PROGRAM PRG_07_Servo
VAR
	fbMC_Power_Ax1: MC_Power;
	fbMC_Power_Ax2: MC_Power;
	fbMC_Jog_Ax1: MC_Jog;
	fbMC_Jog_Ax2: MC_Jog;
	fbMC_Reset_Ax1: MC_Reset;
	fbMC_Reset_Ax2: MC_Reset;
	fbMC_Stop_Ax1: MC_Stop;
	fbMC_Stop_Ax2: MC_Stop;
	
	rJogSpeed:	REAL;
	
	bTest1: BOOL;
	MC_ReadStatus_0: MC_ReadStatus;
	MC_ReadStatus_1: MC_ReadStatus;
	R_TRIG_0: R_TRIG;
	R_TRIG_1: R_TRIG;
	MC_MoveVelocity_0: MC_MoveVelocity;
	uAx1Encoder: UDINT;
	bJogSpeedChange: BOOL;
	t_JogSpeedChange: TP;
	JogSpeegTrig: F_TRIG;
	iPowerOverride: INT;
	tof_SawDownLimit: TOF;
	TRIG_SawDownLimit: r_trig;
	SR_SawDownLimit: SR;

	ton_SawDownLimitTimer: ton;
	SR_ZAxisBuffer: SR;
	F_TRIG_ZAxisCapturedValue: F_TRIG;
	rZAxisBufferSpeed: REAL;
	rZAxisSlowSpeed: REAL;
	rZAxisMedSpeed: REAL;
	rZAxisFastSpeed: REAL;
	sr_ZAxisBufferZone: SR;
	rZAxisCurrentFeedbackSpeed: REAL;
	F_TRIG_ZAxisUpperLimitValue: F_TRIG;
	F_TRIG_ZAxisLowerLimitValue: F_TRIG;
	iZAxisCapturedBufferValue: DINT;

END_VAR

ACTION ACT_07_1_Power:
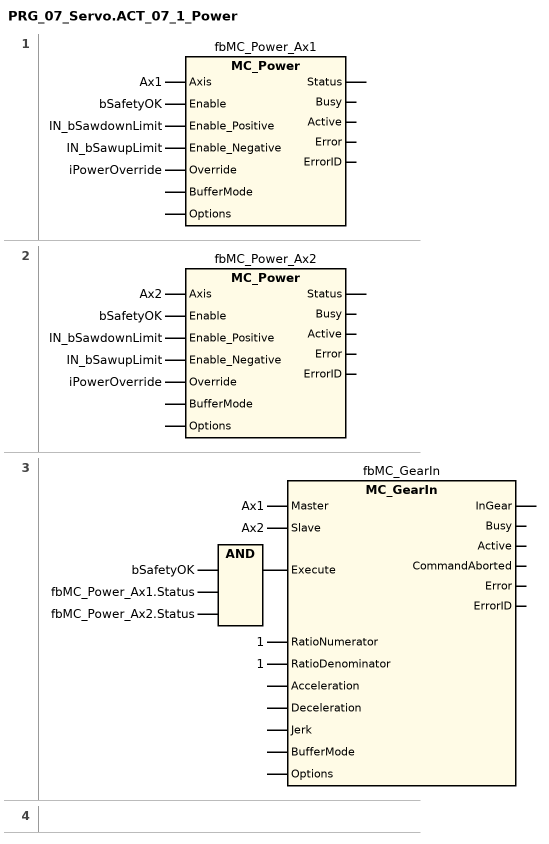
// NETWORK 1
fbMC_Power_Ax1(
    Axis := Ax1,
    Enable := bSafetyOK,
    Enable_Positive := IN_bSawdownLimit,
    Enable_Negative := IN_bSawupLimit,
    Override := iPowerOverride); // MC_Power

// NETWORK 2
fbMC_Power_Ax2(
    Axis := Ax2,
    Enable := bSafetyOK,
    Enable_Positive := IN_bSawdownLimit,
    Enable_Negative := IN_bSawupLimit,
    Override := iPowerOverride); // MC_Power

// NETWORK 3
fbMC_GearIn(
    Master := Ax1,
    Slave := Ax2,
    Execute := bSafetyOK AND fbMC_Power_Ax1.Status AND fbMC_Power_Ax2.Status,
    RatioNumerator := 1,
    RatioDenominator := 1); // MC_GearIn

// NETWORK 4
END_ACTION

ACTION ACT_07_2_Reset:
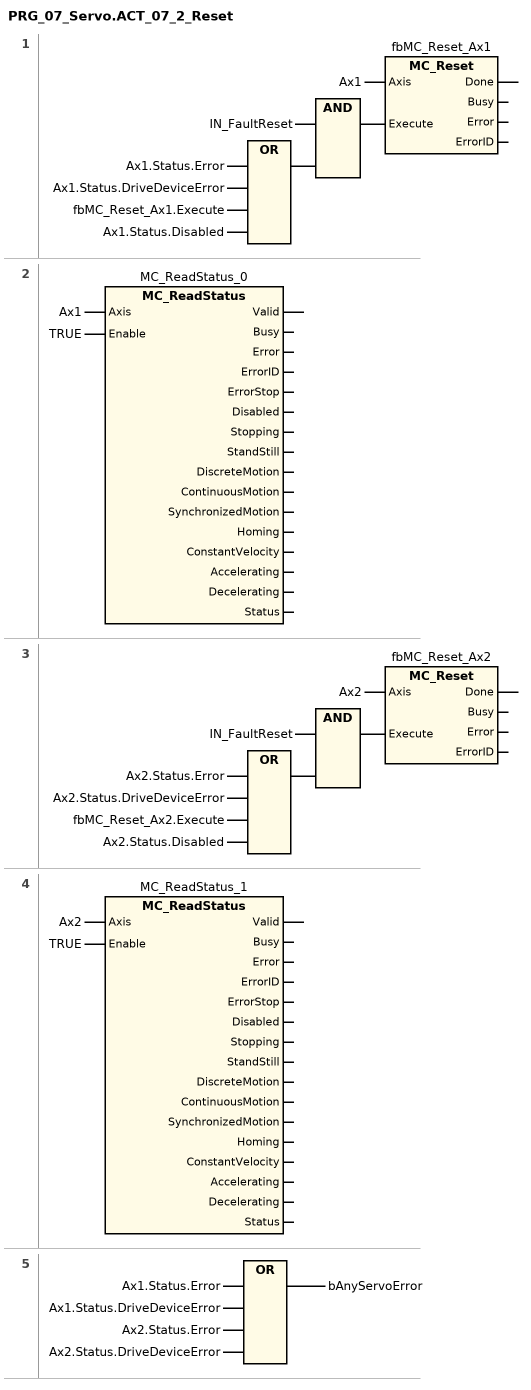
// NETWORK 1
fbMC_Reset_Ax1(Axis := Ax1, Execute := IN_FaultReset AND (Ax1.Status.Error OR Ax1.Status.DriveDeviceError OR fbMC_Reset_Ax1.Execute OR Ax1.Status.Disabled)); // MC_Reset

// NETWORK 2
MC_ReadStatus_0(Axis := Ax1, Enable := TRUE); // MC_ReadStatus

// NETWORK 3
fbMC_Reset_Ax2(Axis := Ax2, Execute := IN_FaultReset AND (Ax2.Status.Error OR Ax2.Status.DriveDeviceError OR fbMC_Reset_Ax2.Execute OR Ax2.Status.Disabled)); // MC_Reset

// NETWORK 4
MC_ReadStatus_1(Axis := Ax2, Enable := TRUE); // MC_ReadStatus

// NETWORK 5
bAnyServoError := Ax1.Status.Error OR Ax1.Status.DriveDeviceError OR Ax2.Status.Error OR Ax2.Status.DriveDeviceError;

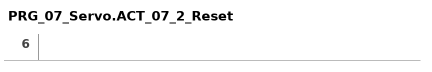
// NETWORK 6
END_ACTION

ACTION ACT_07_3_Jog:
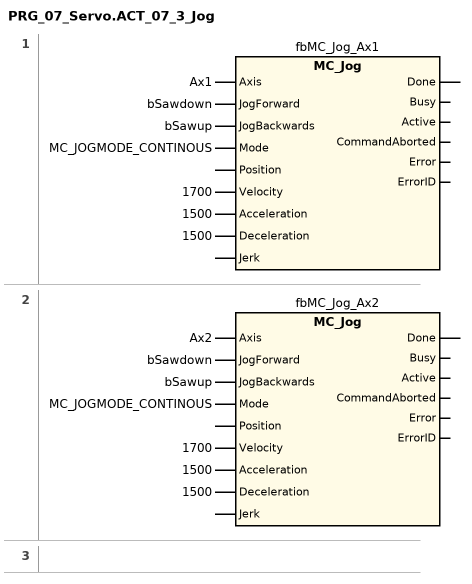
// NETWORK 1
fbMC_Jog_Ax1(
    Axis := Ax1,
    JogForward := bSawdown,
    JogBackwards := bSawup,
    Mode := MC_JOGMODE_CONTINOUS,
    Velocity := 1700,
    Acceleration := 1500,
    Deceleration := 1500); // MC_Jog

// NETWORK 2
fbMC_Jog_Ax2(
    Axis := Ax2,
    JogForward := bSawdown,
    JogBackwards := bSawup,
    Mode := MC_JOGMODE_CONTINOUS,
    Velocity := 1700,
    Acceleration := 1500,
    Deceleration := 1500); // MC_Jog

// NETWORK 3
END_ACTION

ACTION ACT_07_4_JogSpeed:
(* Z-axis speed setpoints *)
rZAxisBufferSpeed 	:= 950 ;
rZAxisSlowSpeed 	:= 1000 ;
rZAxisMedSpeed 		:= 1400 ;
rZAxisFastSpeed 	:= 1700 ;
rZAxisCurrentFeedbackSpeed := 750 ;

(* Z-axis capture value for the buffer zone *)
F_TRIG_ZAxisUpperLimitValue(CLK:= IN_bSawUpLimit, Q=> );
IF bSawUP AND F_TRIG_ZAxisUpperLimitValue.Q THEN
	iZAxisUpperLimitValue := LREAL_TO_DINT(Ax1.NcToPlc.ActPos) ;
END_IF

F_TRIG_ZAxisLowerLimitValue(CLK:= IN_bSawDownLimit, Q=> );
IF F_TRIG_ZAxisLowerLimitValue.Q THEN
	iZAxisLowerLimitValue := LREAL_TO_DINT(Ax1.NcToPlc.ActPos) ;
END_IF

	iZAxisCapturedBufferValue := iZAxisLowerLimitValue - 17040 ;	// approx. 3" high from the bed

(* Z-axis selector switch *)
IF		IN_bZaxisSlow	THEN
		rJogSpeed	:=	rZAxisSlowSpeed	;
ELSIF	IN_bZaxisFAST	THEN
		rJogSpeed	:=	rZAxisFastSpeed	;
ELSE	rJogSpeed	:=	rZAxisMedSpeed	;
END_IF

(* Z-axis power override limit at max 100% and min 0% *)
IF iPowerOverride > 100 THEN
	iPowerOverride := 100 ;
ELSIF iPowerOverride < 0 THEN
	iPowerOverride := 0 ;
END_IF

 (* Z-axis Jog speed *)
IF (Ax1.NcToPlc.ActPos > DINT_TO_LREAL(iZAxisCapturedBufferValue)) AND bSawDOWN AND rCrossCutSpeedMultiplier > 0.75 THEN	
	iPowerOverride := REAL_TO_INT((rZAxisBufferSpeed / rZAxisFastSpeed)*100) ;			// Z-axis buffer zone speed
	
ELSIF bSawDOWN AND rCrossCutSpeedMultiplier <= 0.75 THEN	
	iPowerOverride := REAL_TO_INT((rZAxisCurrentFeedbackSpeed / rZAxisFastSpeed)*100) ;	// Z-axis current feedback speed
	
ELSIF (Ax1.NcToPlc.ActPos >= DINT_TO_LREAL(iZAxisCapturedBufferValue)) AND bSawDOWN AND rCrossCutSpeedMultiplier > 0.75 THEN
	iPowerOverride := REAL_TO_INT((rJogSpeed / rZAxisFastSpeed)*100) ;					// Z-axis speed selector switch
	
ELSIF NOT bSawDOWN OR bSawUP THEN
	iPowerOverride := 100 ;
END_IF
END_ACTION

ACTION ACT_07_5_Stop:
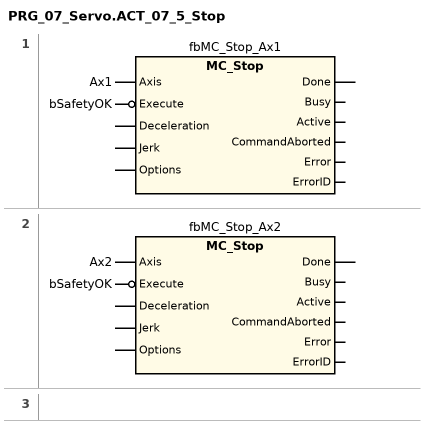
// NETWORK 1
fbMC_Stop_Ax1(Axis := Ax1, Execute := NOT bSafetyOK); // MC_Stop

// NETWORK 2
fbMC_Stop_Ax2(Axis := Ax2, Execute := NOT bSafetyOK); // MC_Stop

// NETWORK 3
END_ACTION

END_PROGRAM

(* stored: Version 1.1.0.1, ProductVersion 3.1.4024.12
   POU PRG_07_Servo: Id {e88641b0-86d9-4b7a-a7c8-72cb56abef6c}, SpecialFunc None
   Action ACT_07_1_Power: Id {42f6af81-1d23-4666-b486-a7bd697e0208}
   Action ACT_07_2_Reset: Id {095d0706-9aec-4af4-8dca-983fa52b58f9}
   Action ACT_07_3_Jog: Id {15f3ce89-87fa-4f3b-865f-d7b9d662b8b3}
   Action ACT_07_4_JogSpeed: Id {ae2b6ce5-0293-4c56-941c-82276bc16f0a}
   Action ACT_07_5_Stop: Id {d29df8b9-f9be-4655-bc9c-1dacf7ece49e} *)
